FUNCTION_BLOCK CU050AutomatParalell_1_Task EXTENDS TcoTaskedSequencer 

VAR
	_customTimer: TON;
END_VAR

Run();

(*~
	<docu>
		<summary>
			Main method of the sequener. Custom code needs to be placed here. The sequencer is executed by call of **Instance.Run()** method.
			This method is abstract, and it must be overridden in derived block.
		</summary>
	</docu>
~*)
METHOD PROTECTED Main : BOOL
// Takes mode (step/continous) from the parent controller
THIS^.ModeController.Mode := ParentSequence.ModeController.Mode;

IF (Step(1000, TRUE, 'PARALELL STEP - EXAMPLE OF TIMERS')) THEN
    //-------------------------------------    
		StepCompleteWhen(CurrentStep.Duration >= T#300mS);	
    //-------------------------------------
END_IF
IF (Step(1100, TRUE, 'PARALELL STEP - EXAMPLE OF TIMERS')) THEN
    //-------------------------------------    
		StepCompleteWhen(inCondition:=Timer_1(TRUE,T#100MS));	
    //-------------------------------------
END_IF
IF (Step(1200, TRUE, 'PARALELL STEP - EXAMPLE OF TIMERS')) THEN
    //-------------------------------------    
		StepCompleteWhen(inCondition:=Timer_1(TRUE,T#200MS));	
    //-------------------------------------
END_IF


IF THIS^.IsFreshState THEN
	_customTimer(IN:=FALSE);
END_IF
IF (Step(1300, TRUE, 'PARALELL STEP - EXAMPLE OF TIMERS')) THEN
    //-------------------------------------    

		_customTimer(IN:=TRUE,PT:=T#200MS);
		StepCompleteWhen(inCondition:=_customTimer.Q);	
    //-------------------------------------
END_IF


IF (Step(10000, TRUE, 'PARALELL TASK DONE')) THEN
    //-------------------------------------
    _task.DoneWhen(TRUE );
    //-------------------------------------	
END_IF
END_METHOD

PROPERTY ParentSequence : REFERENCE TO CU050AutomatTask
GET
VAR
    _parentSequence : POINTER TO CU050AutomatTask;
END_VAR
IF __QUERYPOINTER(Parent, _parentSequence) THEN 
    ParentSequence REF= _parentSequence^;              
END_IF
END_GET
END_PROPERTY

END_FUNCTION_BLOCK

(* stored: Version 1.1.0.1
   POU CU050AutomatParalell_1_Task: Id {538dad44-8454-43fd-9373-4c4444597446}, SpecialFunc None
   Method Main: Id {fee8e497-55d9-4a6d-8585-54a44d2dbec3}
   Property ParentSequence: Id {2cf70b35-7979-4992-b8d6-684130c1d9b0}
   Get Get: Id {af3c1841-730c-4deb-a0fc-b577450c54c1} *)
